// TIA Portal project "2022.04.30—定时器2" (V17)

(* hardware
DEVICE "S7-1500/ET200MP station_1"  S7-1500 station
   slot 0: "导轨_0"  Rack  6ES7 590-1***0-0AA0
   slot 1: "PLC_1"  CPU 1516-3 PN/DP  6ES7 516-3AN00-0AB0  V1.7
      slot 3: "CPU 显示_1"  6ES7591-1BA00-0AA0
      slot 32768: "PROFINET 接口_1"  X1
         slot 32769: "端口_1"  X1 P1
         slot 32770: "端口_2"  X1 P2
      slot 33024: "PROFINET 接口_2"  X2
         slot 33025: "端口_1"  X2 P1
      slot 33280: "DP 接口_1"  X3
   slot 2: "DI 32x24VDC BA_1"  DI 32x24VDC BA  6ES7 521-1BL10-0AA0  V1.1
   slot 3: "DQ 32x24VDC/0.5A HF_1"  DQ 32x24VDC/0.5A HF  6ES7 522-1BL01-0AB0  V1.1
*)

// ===== PLC "PLC_1"  CPU 1516-3 PN/DP =====

VAR_GLOBAL   // PLC tag table "默认变量表"
   "按钮1" AT %I0.0 : Bool;
   "按钮2" AT %I0.1 : Bool;
   "按钮3" AT %I0.2 : Bool;
   "按钮4" AT %I0.3 : Bool;
   "按钮5" AT %I0.4 : Bool;
   "按钮6" AT %I0.5 : Bool;
   "按钮7" AT %I0.6 : Bool;
   "按钮8" AT %I0.7 : Bool;
   "按钮9" AT %I1.0 : Bool;
   "按钮10" AT %I1.1 : Bool;
   "按钮11" AT %I1.2 : Bool;
   "指示灯1" AT %Q0.0 : Bool;
   "指示灯2" AT %Q0.1 : Bool;
   "指示灯3" AT %Q0.2 : Bool;
   "指示灯4" AT %Q0.3 : Bool;
   "指示灯5" AT %Q0.4 : Bool;
   "指示灯6" AT %Q0.5 : Bool;
   "指示灯7" AT %Q0.6 : Bool;
   "指示灯8" AT %Q0.7 : Bool;
   "指示灯9" AT %Q1.0 : Bool;
   "指示灯10" AT %Q1.1 : Bool;
   "指示灯11" AT %Q1.2 : Bool;
   "指示灯12" AT %Q1.3 : Bool;
   "1" AT %M1.0 : Bool;
   "0" AT %M1.1 : Bool;
   "Tag_1" AT %M0.1 : Bool;
   "Tag_3" AT %T1 : Timer;
   "Tag_4" AT %T2 : Timer;
   "Tag_5" AT %T3 : Timer;
   "Tag_6" AT %T4 : Timer;
   "Tag_7" AT %T6 : Timer;
   "Tag_8" AT %M50.0 : Bool;
   "Tag_2" AT %T8 : Timer;
END_VAR

DATA_BLOCK "计数器LCD_DB"   // DB2
{ S7_Optimized_Access := 'TRUE' }
VERSION : 0.1
// stored: InstanceOfName 计数器LCD
"计数器LCD"
BEGIN
END_DATA_BLOCK

DATA_BLOCK "定时器DB"   // DB3
{ S7_Optimized_Access := 'TRUE' }
VERSION : 0.1
   VAR
      老版定时器 : Struct
         分配关断延时定时器并启动_q : Bool;
         分配关断延时定时器并启动_bl : Word;
         分配关断延时定时器并启动_BCD_1 : Word;
         分配接通延时定时器并启动_BCD : Word;
         分配接通延时定时器并启动_q : Bool;
         分配接通延时定时器并启动_bl : Word;
         分配脉冲扩展定时器并启动_bl : Word;
         分配脉冲扩展定时器并启动_q : Bool;
         分配脉冲扩展定时器并启动_BCD : Word;
         分配脉冲定时器并启动_BCD : Word;
         分配脉冲定时器并启动_bl : Word;
         分配脉冲定时器并启动_q : Bool;
      END_STRUCT;
      时间累加器 : IEC_TIMER;
      起动关断延时定时器 : IEC_TIMER;
      Static_1 : IEC_TIMER;
      起动接通延时定时器 : IEC_TIMER;
      启动脉冲定时器 : IEC_TIMER;
   END_VAR
BEGIN
END_DATA_BLOCK

DATA_BLOCK "定时器FBD_DB"   // DB4
{ S7_Optimized_Access := 'TRUE' }
VERSION : 0.1
// stored: InstanceOfName 定时器FBD
"定时器FBD"
BEGIN
END_DATA_BLOCK

DATA_BLOCK "定时器SCL_DB"   // DB5
{ S7_Optimized_Access := 'TRUE' }
VERSION : 0.1
// stored: InstanceOfName 定时器SCL
"定时器SCL"
BEGIN
END_DATA_BLOCK

// folder: System blocks/Program resources

DATA_BLOCK "IEC_Timer_0_DB"   // DB1
{ S7_Optimized_Access := 'TRUE' }
AUTHOR : Simatic
FAMILY : IEC
NAME : IEC_TMR
VERSION : 1.0
// stored: InstanceOfName IEC_TIMER
"IEC_TIMER"
BEGIN
END_DATA_BLOCK

// folder: (top level)

FUNCTION_BLOCK "计数器LCD"   // FB1, LAD
{ S7_Optimized_Access := 'TRUE' }
VERSION : 0.1
   VAR
      qq : DInt;
      AA : DInt;
      "A" : DInt;
      生成脉冲_ET : DInt;
      老版定时器 : Struct
      END_STRUCT;
      生成脉冲 : TP_TIME;
      接通延时 : TON_TIME;
      关断延时 : TOF_TIME;
      时间累加 : TONR_TIME;
   END_VAR
   VAR_TEMP   // added for the SCL form of the ladder/FBD networks
      _w1 : Bool;
   END_VAR
BEGIN

REGION Network 1: 按多长时间，就生成多少脉冲
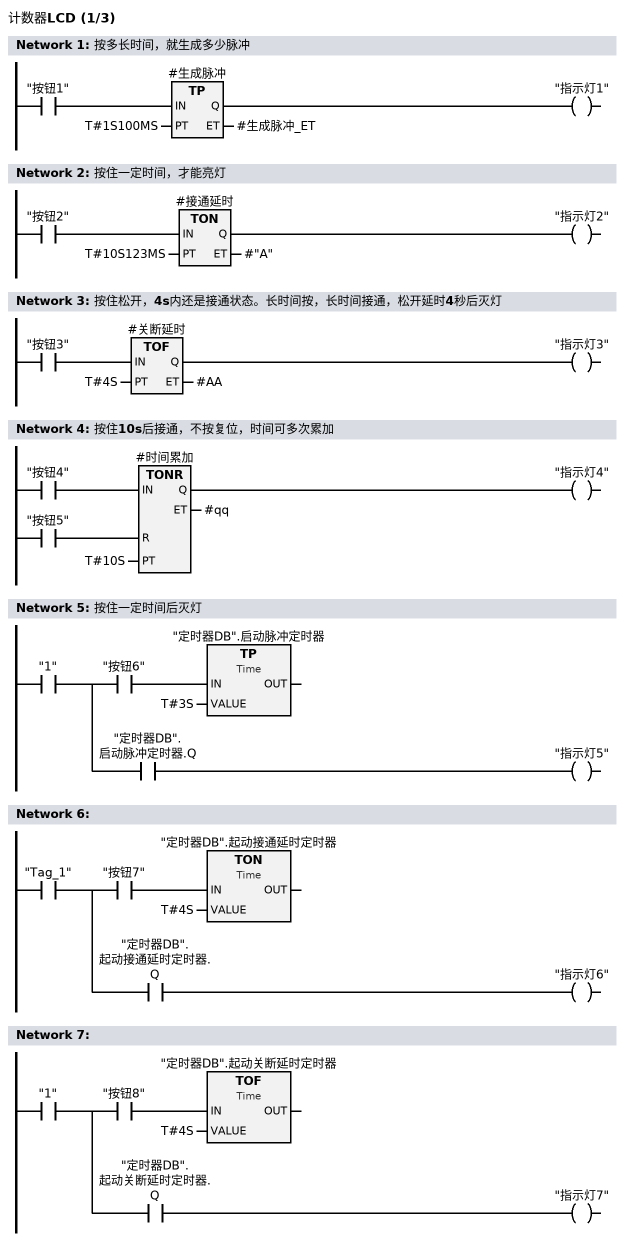
   #生成脉冲(IN := "按钮1", PT := T#1S100MS, ET => #生成脉冲_ET);   // TP
   "指示灯1" := #生成脉冲.Q;
END_REGION

REGION Network 2: 按住一定时间，才能亮灯
   #接通延时(IN := "按钮2", PT := T#10S123MS, ET => #"A");   // TON
   "指示灯2" := #接通延时.Q;
END_REGION

REGION Network 3: 按住松开，4s内还是接通状态。长时间按，长时间接通，松开延时4秒后灭灯
   #关断延时(IN := "按钮3", PT := T#4S, ET => #AA);   // TOF
   "指示灯3" := #关断延时.Q;
END_REGION

REGION Network 4: 按住10s后接通，不按复位，时间可多次累加
   #时间累加(IN := "按钮4", R := "按钮5", PT := T#10S, ET => #qq);   // TONR
   "指示灯4" := #时间累加.Q;
END_REGION

REGION Network 5: 按住一定时间后灭灯
   "定时器DB".启动脉冲定时器.TP(IN := "1" AND "按钮6", PT := T#3S);   // TP coil
   "指示灯5" := "1" AND "定时器DB".启动脉冲定时器.Q;
END_REGION

REGION Network 6
   "定时器DB".起动接通延时定时器.TON(IN := "Tag_1" AND "按钮7", PT := T#4S);   // TON coil
   "指示灯6" := "Tag_1" AND "定时器DB".起动接通延时定时器.Q;
END_REGION

REGION Network 7
   "定时器DB".起动关断延时定时器.TOF(IN := "1" AND "按钮8", PT := T#4S);   // TOF coil
   "指示灯7" := "1" AND "定时器DB".起动关断延时定时器.Q;
END_REGION

REGION Network 8
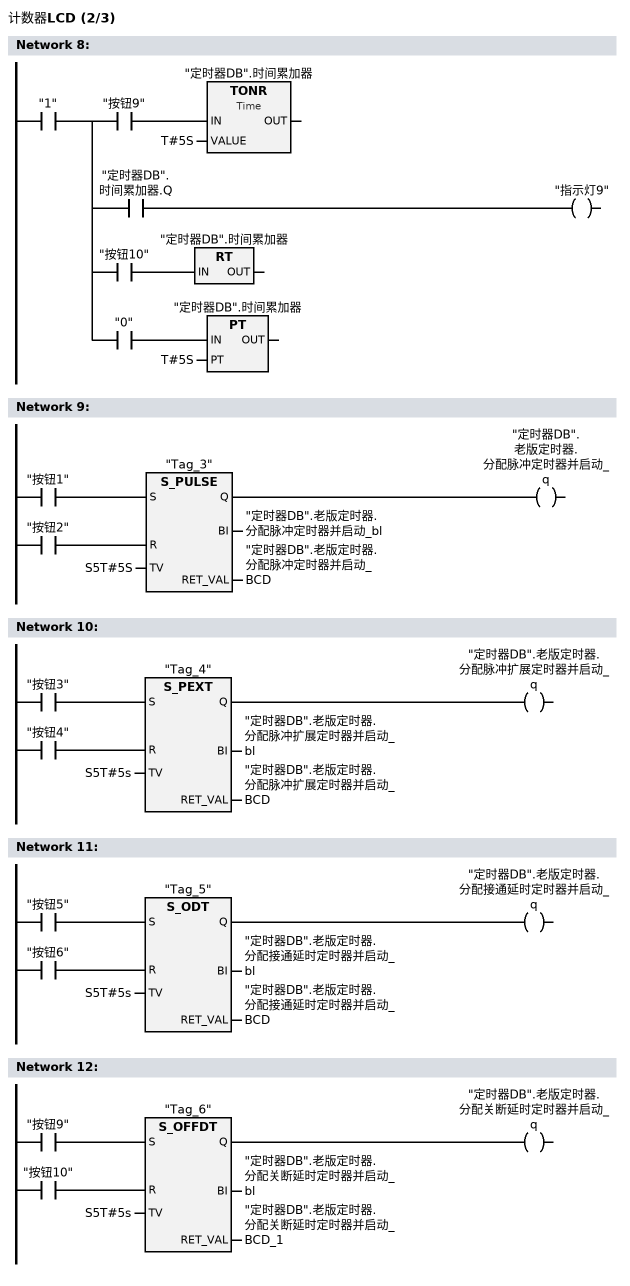
   "定时器DB".时间累加器.TONR(IN := "1" AND "按钮9", PT := T#5S);   // TONR coil
   "指示灯9" := "1" AND "定时器DB".时间累加器.Q;
   IF "1" AND "按钮10" THEN RESET_TIMER("定时器DB".时间累加器); END_IF;
   IF "1" AND "0" THEN PRESET_TIMER(PT := T#5S, TIMER := "定时器DB".时间累加器); END_IF;
END_REGION

REGION Network 9
   RUNG wire#powerrail
      Contact( "按钮1" )
      S_PULSE(T_NO := "Tag_3", R := wire#w1, TV := S5T#5S, BI => "定时器DB".老版定时器.分配脉冲定时器并启动_bl, RET_VAL => "定时器DB".老版定时器.分配脉冲定时器并启动_BCD)
      Coil( "定时器DB".老版定时器.分配脉冲定时器并启动_q )
   END_RUNG
   RUNG wire#powerrail
      Contact( "按钮2" )
   END_RUNG wire#w1
   // the same network as SCL:
   "定时器DB".老版定时器.分配脉冲定时器并启动_BCD := S_PULSE(T_NO := "Tag_3",
                           S := "按钮1",
                           R := "按钮2",
                           TV := S5T#5S,
                           Q => #_w1,
                           BI => "定时器DB".老版定时器.分配脉冲定时器并启动_bl);
   "定时器DB".老版定时器.分配脉冲定时器并启动_q := #_w1;
END_REGION

REGION Network 10
   RUNG wire#powerrail
      Contact( "按钮3" )
      S_PEXT(T_NO := "Tag_4", R := wire#w1, TV := S5T#5s, BI => "定时器DB".老版定时器.分配脉冲扩展定时器并启动_bl, RET_VAL => "定时器DB".老版定时器.分配脉冲扩展定时器并启动_BCD)
      Coil( "定时器DB".老版定时器.分配脉冲扩展定时器并启动_q )
   END_RUNG
   RUNG wire#powerrail
      Contact( "按钮4" )
   END_RUNG wire#w1
   // the same network as SCL:
   "定时器DB".老版定时器.分配脉冲扩展定时器并启动_BCD := S_PEXT(T_NO := "Tag_4",
                           S := "按钮3",
                           R := "按钮4",
                           TV := S5T#5s,
                           Q => #_w1,
                           BI => "定时器DB".老版定时器.分配脉冲扩展定时器并启动_bl);
   "定时器DB".老版定时器.分配脉冲扩展定时器并启动_q := #_w1;
END_REGION

REGION Network 11
   RUNG wire#powerrail
      Contact( "按钮5" )
      S_ODT(T_NO := "Tag_5", R := wire#w1, TV := S5T#5s, BI => "定时器DB".老版定时器.分配接通延时定时器并启动_bl, RET_VAL => "定时器DB".老版定时器.分配接通延时定时器并启动_BCD)
      Coil( "定时器DB".老版定时器.分配接通延时定时器并启动_q )
   END_RUNG
   RUNG wire#powerrail
      Contact( "按钮6" )
   END_RUNG wire#w1
   // the same network as SCL:
   "定时器DB".老版定时器.分配接通延时定时器并启动_BCD := S_ODT(T_NO := "Tag_5",
                           S := "按钮5",
                           R := "按钮6",
                           TV := S5T#5s,
                           Q => #_w1,
                           BI => "定时器DB".老版定时器.分配接通延时定时器并启动_bl);
   "定时器DB".老版定时器.分配接通延时定时器并启动_q := #_w1;
END_REGION

REGION Network 12
   RUNG wire#powerrail
      Contact( "按钮9" )
      S_OFFDT(T_NO := "Tag_6", R := wire#w1, TV := S5T#5s, BI => "定时器DB".老版定时器.分配关断延时定时器并启动_bl, RET_VAL => "定时器DB".老版定时器.分配关断延时定时器并启动_BCD_1)
      Coil( "定时器DB".老版定时器.分配关断延时定时器并启动_q )
   END_RUNG
   RUNG wire#powerrail
      Contact( "按钮10" )
   END_RUNG wire#w1
   // the same network as SCL:
   "定时器DB".老版定时器.分配关断延时定时器并启动_BCD_1 := S_OFFDT(T_NO := "Tag_6",
                           S := "按钮9",
                           R := "按钮10",
                           TV := S5T#5s,
                           Q => #_w1,
                           BI => "定时器DB".老版定时器.分配关断延时定时器并启动_bl);
   "定时器DB".老版定时器.分配关断延时定时器并启动_q := #_w1;
END_REGION

REGION Network 13
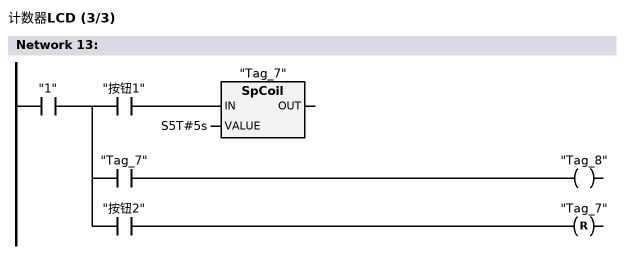
   // no SCL statement known for SpCoil: written as a call
   #_w1 := "1";
   SpCoil(in := "1" AND "按钮1", value := S5T#5s, operand := "Tag_7");
   "Tag_8" := #_w1 AND "Tag_7";
   IF #_w1 AND "按钮2" THEN "Tag_7" := FALSE; END_IF;
END_REGION
END_FUNCTION_BLOCK

FUNCTION_BLOCK "定时器FBD"   // FB2, FBD
{ S7_Optimized_Access := 'TRUE' }
VERSION : 0.1
   VAR
      qq : DInt := 0;
      AA : DInt := 0;
      "A" : DInt := 0;
      生成脉冲_ET : DInt := 0;
      生成脉冲 : TP_TIME;
      接通延时 : TON_TIME;
      关断延时 : TOF_TIME;
      时间累加 : TONR_TIME;
      Static_1 : TP_TIME;
      Static_2 : TON_TIME;
      Static_3 : TOF_TIME;
      Static_4 : TONR_TIME;
   END_VAR
   VAR_TEMP   // added for the SCL form of the ladder/FBD networks
      _w1 : Bool;
   END_VAR
BEGIN

REGION Network 1
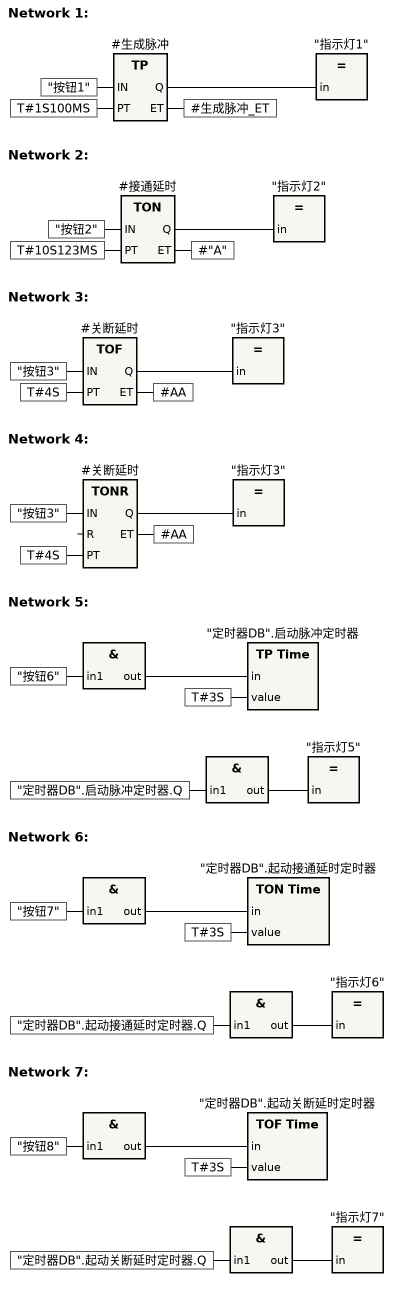
   #生成脉冲(IN := "按钮1", PT := T#1S100MS, ET => #生成脉冲_ET);   // TP
   "指示灯1" := #生成脉冲.Q;
END_REGION

REGION Network 2
   #接通延时(IN := "按钮2", PT := T#10S123MS, ET => #"A");   // TON
   "指示灯2" := #接通延时.Q;
END_REGION

REGION Network 3
   #关断延时(IN := "按钮3", PT := T#4S, ET => #AA);   // TOF
   "指示灯3" := #关断延时.Q;
END_REGION

REGION Network 4
   #关断延时(IN := "按钮3", PT := T#4S, ET => #AA);   // TONR
   "指示灯3" := #关断延时.Q;
END_REGION

REGION Network 5
   "定时器DB".启动脉冲定时器.TP(IN := "按钮6", PT := T#3S);   // TP coil
   "指示灯5" := "定时器DB".启动脉冲定时器.Q;
END_REGION

REGION Network 6
   "定时器DB".起动接通延时定时器.TON(IN := "按钮7", PT := T#3S);   // TON coil
   "指示灯6" := "定时器DB".起动接通延时定时器.Q;
END_REGION

REGION Network 7
   "定时器DB".起动关断延时定时器.TOF(IN := "按钮8", PT := T#3S);   // TOF coil
   "指示灯7" := "定时器DB".起动关断延时定时器.Q;
END_REGION

REGION Network 8
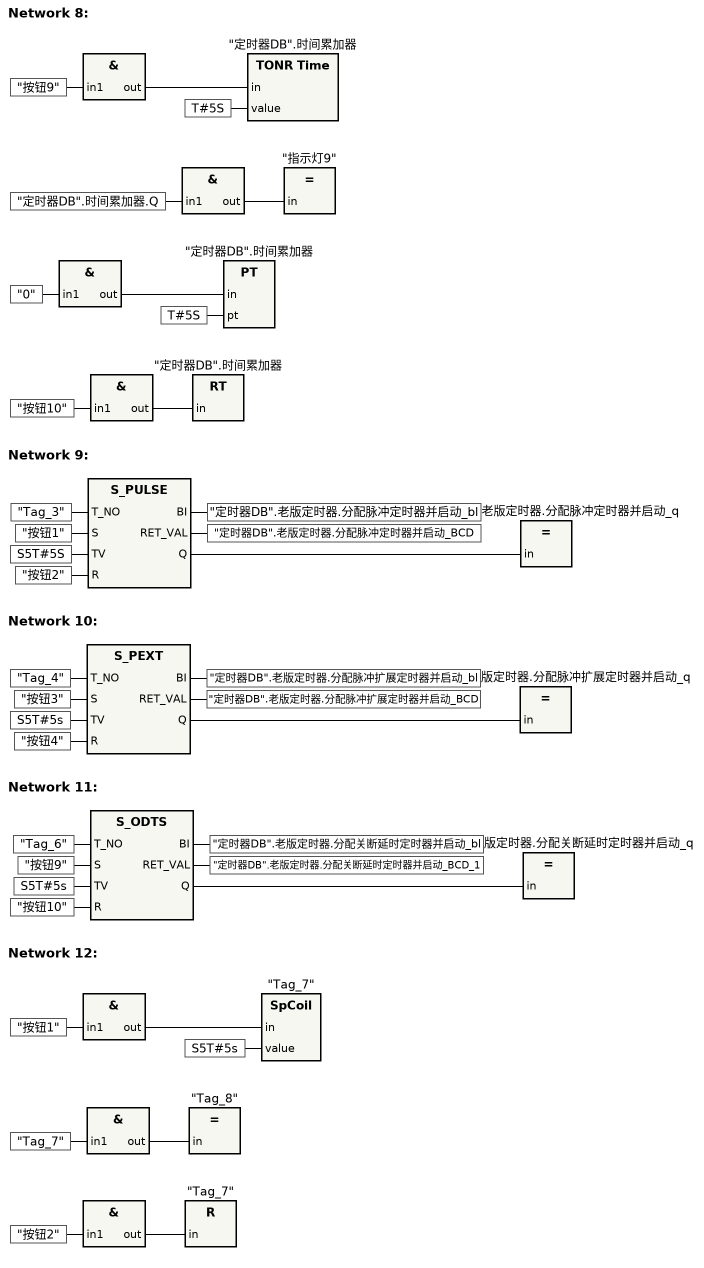
   "定时器DB".时间累加器.TONR(IN := "按钮9", PT := T#5S);   // TONR coil
   "指示灯9" := "定时器DB".时间累加器.Q;
   IF "0" THEN PRESET_TIMER(PT := T#5S, TIMER := "定时器DB".时间累加器); END_IF;
   IF "按钮10" THEN RESET_TIMER("定时器DB".时间累加器); END_IF;
END_REGION

REGION Network 9
   "定时器DB".老版定时器.分配脉冲定时器并启动_BCD := S_PULSE(T_NO := "Tag_3",
                           S := "按钮1",
                           TV := S5T#5S,
                           R := "按钮2",
                           BI => "定时器DB".老版定时器.分配脉冲定时器并启动_bl,
                           Q => #_w1);
   "定时器DB".老版定时器.分配脉冲定时器并启动_q := #_w1;
END_REGION

REGION Network 10
   "定时器DB".老版定时器.分配脉冲扩展定时器并启动_BCD := S_PEXT(T_NO := "Tag_4",
                           S := "按钮3",
                           TV := S5T#5s,
                           R := "按钮4",
                           BI => "定时器DB".老版定时器.分配脉冲扩展定时器并启动_bl,
                           Q => #_w1);
   "定时器DB".老版定时器.分配脉冲扩展定时器并启动_q := #_w1;
END_REGION

REGION Network 11
   "定时器DB".老版定时器.分配关断延时定时器并启动_BCD_1 := S_ODTS(T_NO := "Tag_6",
                           S := "按钮9",
                           TV := S5T#5s,
                           R := "按钮10",
                           BI => "定时器DB".老版定时器.分配关断延时定时器并启动_bl,
                           Q => #_w1);
   "定时器DB".老版定时器.分配关断延时定时器并启动_q := #_w1;
END_REGION

REGION Network 12
   // no SCL statement known for SpCoil: written as a call
   SpCoil(in := "按钮1", value := S5T#5s, operand := "Tag_7");
   "Tag_8" := "Tag_7";
   IF "按钮2" THEN "Tag_7" := FALSE; END_IF;
END_REGION
END_FUNCTION_BLOCK

FUNCTION_BLOCK "定时器SCL"   // FB3, SCL
{ S7_Optimized_Access := 'TRUE' }
VERSION : 0.1
   VAR
      IEC_Timer_0_Instance : TP_TIME;
      IEC_Timer_0_Instance_1 : TON_TIME;
      IEC_Timer_0_Instance_2 : TOF_TIME;
      IEC_Timer_0_Instance_3 : TONR_TIME;
   END_VAR
BEGIN
   #生成脉冲(IN:="按钮1",
                         PT:=T#1S100MS,
                         Q=>"指示灯1",
                         ET=>#生成脉冲_ET);

    #IEC_Timer_0_Instance_1(IN:="按钮2",
                            PT:=T#10S123MS,
                            Q=>"指示灯2",
                            ET=>#A);

   #IEC_Timer_0_Instance_2(IN:="按钮3",
                           PT:=T#4S,
                           Q=>"指示灯3",
                           ET=>#AA);

   IF "按钮8" THEN
       RESET_TIMER(#IEC_Timer_0_Instance_3);
   END_IF;

   IF "0" THEN
       RESET_TIMER(PT := time_in,
                   TIMER := #IEC_Timer_0_Instance_3);
   END_IF;

   #IEC_Timer_0_Instance_3(IN:="按钮4",
                           R:="按钮5",
                           PT:=T#10S,
                           Q=>"指示灯4",
                           ET=>#qq);

   "定时器DB".老版定时器.分配脉冲定时器并启动_BCD:=S_PULSE(T_NO := "Tag_3",
           S := "按钮1",
           TV := S5T#5S,
           R := "按钮2",
           BI => "定时器DB".老版定时器.分配脉冲定时器并启动_bl,
           Q => "定时器DB".老版定时器.分配脉冲定时器并启动_q);

   "定时器DB".老版定时器.分配脉冲扩展定时器并启动_BCD:=S_PEXT(T_NO := "Tag_4",
          S := "按钮3",
          TV := S5T#5s,
          R := "按钮4",
          BI => "定时器DB".老版定时器.分配脉冲扩展定时器并启动_bl,
          Q => "定时器DB".老版定时器.分配脉冲扩展定时器并启动_q);
END_FUNCTION_BLOCK

ORGANIZATION_BLOCK "Main"   // OB1, LAD, ProgramCycle
TITLE = "Main Program Sweep (Cycle)"
{ S7_Optimized_Access := 'TRUE' }
VERSION : 0.1
   VAR_INPUT
      Initial_Call : Bool;   // Initial call of this OB
      Remanence : Bool;   // =True, if remanent data are available
   END_VAR
BEGIN

REGION Network 1: 1
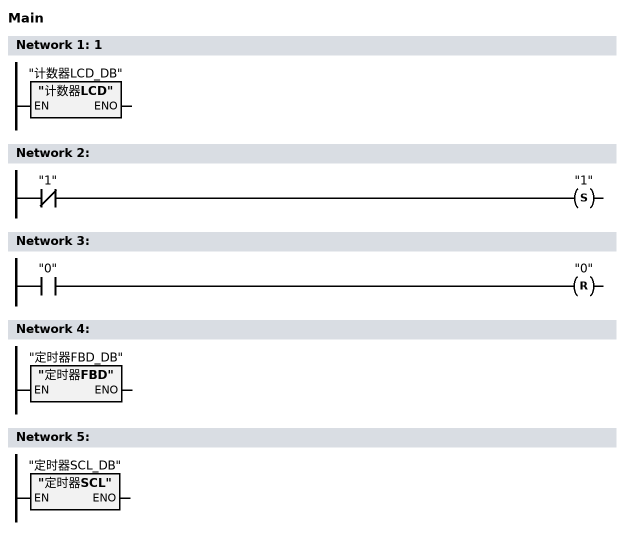
   RUNG wire#powerrail
      "计数器LCD_DB"()
   END_RUNG
   // the same network as SCL:
   "计数器LCD_DB"();   // "计数器LCD"
END_REGION

REGION Network 2
   RUNG wire#powerrail
      I_Contact( "1" )
      S_Coil( "1" )
   END_RUNG
   // the same network as SCL:
   IF NOT "1" THEN "1" := TRUE; END_IF;
END_REGION

REGION Network 3
   RUNG wire#powerrail
      Contact( "0" )
      R_Coil( "0" )
   END_RUNG
   // the same network as SCL:
   IF "0" THEN "0" := FALSE; END_IF;
END_REGION

REGION Network 4
   RUNG wire#powerrail
      "定时器FBD_DB"()
   END_RUNG
   // the same network as SCL:
   "定时器FBD_DB"();   // "定时器FBD"
END_REGION

REGION Network 5
   RUNG wire#powerrail
      "定时器SCL_DB"()
   END_RUNG
   // the same network as SCL:
   "定时器SCL_DB"();   // "定时器SCL"
END_REGION
END_ORGANIZATION_BLOCK